Staubli VAL3: onF8Event.pgx

program onF8Event()
  local num i
  local num l_nResult
 begin
  // look if the bButton is enable
  if bButton[7]
    //
    call use:timerDialog("数据正在保存中....",1)
    call cycle:save(l_nResult)
    if l_nResult==0
      call use:timerDialog("数据已经保存成功",1)
    elseIf l_nResult!=0
      call use:timerDialog("数据未保存成功",1)
    endIf
  endIf
end
